Universal Robots PolyScope program: wrs2020_taskboard_belt.urp

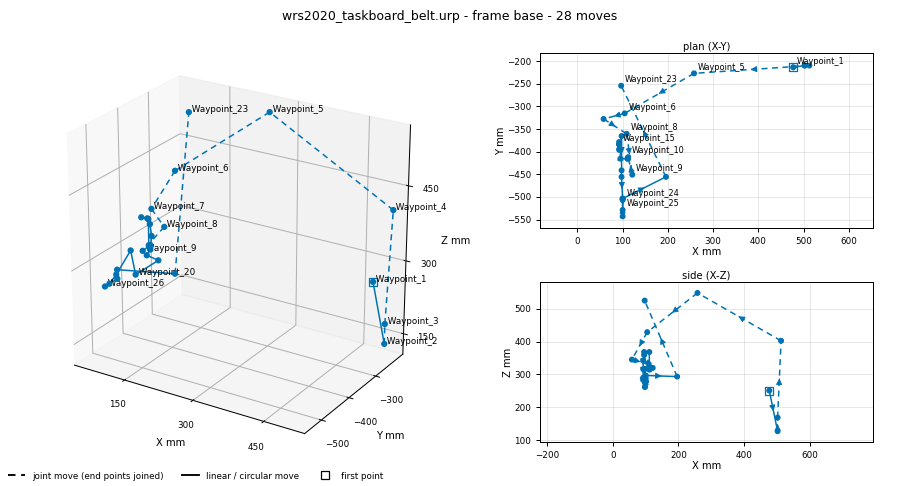
[picture p0: tool path of wrs2020_taskboard_belt.urp in frame base, 28 of 28 moves have a stored position in this frame; points joined in program order, loops and branches not executed]
Program wrs2020_taskboard_belt (installation=default directory=/programs/usbdisk createdIn=3.8.0.61336 lastSavedIn=3.8.0.61336 robotSerialNumber=2018357778)
Calibrated DH parameters: a=[0.000041, -0.391787, -0.374281, -0.000186, 0.000127, 0]; d=[0.08944, 27.652986, -9.436013, -18.1067, 0.094919, 0.082633]; alpha=[1.569511, -0.005996, -0.006449, 1.570544, -1.570475, 0]; deltaTheta=[0.000024, -0.400349, 0.096271, 0.298279, -0.00003, 0.000025]
Robot Program (runOnlyOnce=true)
  URCap Gripper (Robotiq_Grippers, Robotiq Inc.) dataModel(position=0.0, force=100.0, speed=100.0, positionInDouble=0.0, forceInDouble=100.0, speedInDouble=100.0, slaveIds=[9], blocking=true)
  MoveJ speed 60 deg/s, acceleration 80 deg/s^2 (useActiveTCP=true)
    Waypoint Waypoint_1: TCP in base x=476.88 y=-213.476 z=250.862 mm, rx=1.6793 ry=-1.6521 rz=-0.7958 rad; joints [147.47, -71.594, 89.892, -60.74, -116.873, 338.983] deg
  MoveL speed 250 mm/s, acceleration 1200 mm/s^2 (useActiveTCP=true) feature=Base
    Waypoint Waypoint_2: TCP in base x=502.313 y=-209.586 z=126.998 mm, rx=1.6772 ry=-1.66 rz=-0.8065 rad; joints [149.034, -61.436, 94.891, -75.152, -115.221, 340.261] deg
    URCap Gripper (Robotiq_Grippers, Robotiq Inc.) dataModel(position=100.0, force=100.0, speed=100.0, positionInDouble=100.0, forceInDouble=100.0, speedInDouble=100.0, slaveIds=[9], blocking=true)
  MoveJ speed 60 deg/s, acceleration 80 deg/s^2 (useActiveTCP=true)
    Waypoint Waypoint_3: TCP in base x=502.291 y=-209.619 z=168.566 mm, rx=1.6772 ry=-1.6602 rz=-0.8062 rad; joints [149.028, -64.302, 92.335, -69.737, -115.191, 340.279] deg
    Waypoint Waypoint_4: TCP in base x=512.821 y=-209.633 z=402.821 mm, rx=2.1959 ry=-2.1936 rz=-0.0165 rad; joints [146.25, -82.062, 85.641, -92.195, -92.332, 326.65] deg
    Waypoint Waypoint_5: TCP in base x=257.912 y=-226.881 z=548.602 mm, rx=-2.252 ry=-2.1409 rz=0.0571 rad; joints [120.027, -108.226, 87.388, -67.4, -92.623, 123.461] deg
    Popup Message (haltProgram=false message=waiting for a_bot to hold belt inputType=Text)
  MoveJ speed 60 deg/s, acceleration 80 deg/s^2 (useActiveTCP=true)
    Waypoint Waypoint_6: TCP in base x=104.652 y=-315.264 z=429.034 mm, rx=-0.7232 ry=-2.7798 rz=0.8385 rad; joints [93.055, -116.851, 119.471, -121.466, -107.654, 27.881] deg
    Waypoint Waypoint_7: TCP in base x=58.057 y=-327.656 z=345.432 mm, rx=-0.943 ry=-2.6822 rz=1.0186 rad; joints [84.311, -114.161, 133.07, -146.038, -105.388, 27.982] deg
  Popup Message (haltProgram=false message=wait for a_bot to move closer to pulley inputType=Text)
  MoveJ speed 60 deg/s, acceleration 80 deg/s^2 (useActiveTCP=true)
    Waypoint Waypoint_8: TCP in base x=109.129 y=-360.526 z=332.009 mm, rx=-1.6529 ry=-2.3933 rz=0.9597 rad; joints [95.219, -105.447, 127.131, -138.287, -116.294, 68.286] deg
    Waypoint Waypoint_9: TCP in base x=121.477 y=-450.838 z=319.976 mm, rx=-1.9847 ry=-2.0091 rz=0.7379 rad; joints [96.381, -91.245, 112.208, -119.67, -121.006, 93.458] deg
    Waypoint Waypoint_10: TCP in base x=112.095 y=-412.15 z=315.009 mm, rx=-1.9566 ry=-2.0028 rz=0.6969 rad; joints [95.734, -96.48, 117.235, -117.427, -121.063, 92.728] deg
  Popup Message (haltProgram=false message=wait for a_bot to finish placement inputType=Text)
  MoveL speed 250 mm/s, acceleration 1200 mm/s^2 (useActiveTCP=true) feature=Base
    Waypoint Waypoint_11: TCP in base x=111.067 y=-415.408 z=315.577 mm, rx=-1.9655 ry=-2.0043 rz=0.7162 rad; joints [95.563, -96.141, 117.17, -118.803, -121.129, 92.461] deg
    Waypoint Waypoint_12: TCP in base x=111.014 y=-415.438 z=368.385 mm, rx=-1.9655 ry=-2.004 rz=0.716 rad; joints [95.529, -98.391, 111.022, -110.38, -121.122, 92.491] deg
    Waypoint Waypoint_13: TCP in base x=95.213 y=-415.423 z=368.401 mm, rx=-1.9654 ry=-2.0041 rz=0.7161 rad; joints [93.34, -99.062, 111.894, -111.876, -120.787, 89.955] deg
    Waypoint Waypoint_14: TCP in base x=95.201 y=-395.921 z=359.198 mm, rx=-1.9656 ry=-2.0041 rz=0.7161 rad; joints [93.52, -101.499, 115.201, -112.651, -120.798, 90.156] deg
    Waypoint Waypoint_15: TCP in base x=92.395 y=-383.717 z=342.34 mm, rx=-1.9656 ry=-2.0041 rz=0.7163 rad; joints [93.226, -102.722, 118.728, -115.146, -120.743, 89.794] deg
    Waypoint Waypoint_16: TCP in base x=92.424 y=-378.74 z=316.285 mm, rx=-1.9655 ry=-2.0042 rz=0.7161 rad; joints [93.292, -102.186, 122.322, -119.247, -120.747, 89.837] deg
    Waypoint Waypoint_17: TCP in base x=92.37 y=-383.706 z=290.126 mm, rx=-1.9656 ry=-2.0041 rz=0.716 rad; joints [93.254, -99.843, 124.649, -123.945, -120.746, 89.776] deg
    Waypoint Waypoint_18: TCP in base x=92.376 y=-395.73 z=283.079 mm, rx=-1.9656 ry=-2.0041 rz=0.7161 rad; joints [93.151, -97.601, 123.978, -125.581, -120.74, 89.651] deg
    Waypoint Waypoint_19: TCP in base x=97.787 y=-365.382 z=262.233 mm, rx=-2.0667 ry=-2.0015 rz=0.9366 rad; joints [94.505, -99.478, 132.408, -142.318, -121.782, 90.846] deg
    Waypoint Waypoint_20: TCP in base x=97.788 y=-441.256 z=262.195 mm, rx=-2.0667 ry=-2.0016 rz=0.9364 rad; joints [93.65, -88.834, 122.921, -143.961, -121.543, 89.903] deg
    Waypoint Waypoint_21: TCP in base x=97.738 y=-455.581 z=316.933 mm, rx=-2.0668 ry=-2.0015 rz=0.9366 rad; joints [93.494, -91.095, 116.007, -134.854, -121.51, 89.794] deg
  MoveL speed 250 mm/s, acceleration 1200 mm/s^2 (useActiveTCP=true) feature=Base
    Waypoint Waypoint_24: TCP in base x=100.161 y=-506.631 z=288.366 mm, rx=-2.0669 ry=-2.0015 rz=0.9367 rad; joints [93.397, -82.486, 111.528, -139.056, -121.514, 89.661] deg
    Waypoint Waypoint_25: TCP in base x=100.189 y=-528.806 z=278.635 mm, rx=-2.0669 ry=-2.0015 rz=0.9367 rad; joints [93.244, -79.049, 109.068, -140.126, -121.477, 89.482] deg
    Waypoint Waypoint_26: TCP in base x=100.139 y=-542.854 z=278.562 mm, rx=-2.0669 ry=-2.0014 rz=0.9366 rad; joints [93.146, -77.333, 106.94, -139.76, -121.459, 89.381] deg
    Waypoint Waypoint_27: TCP in base x=100.153 y=-503.541 z=278.632 mm, rx=-2.0669 ry=-2.0013 rz=0.9368 rad; joints [93.423, -82.168, 112.794, -140.632, -121.525, 89.684] deg
    Waypoint Waypoint_28: TCP in base x=100.159 y=-503.538 z=296.982 mm, rx=-2.0669 ry=-2.0014 rz=0.9367 rad; joints [93.417, -83.468, 111.222, -137.751, -121.523, 89.695] deg
  MoveL speed 250 mm/s, acceleration 1200 mm/s^2 (useActiveTCP=true) feature=Base
    Waypoint Waypoint_22: TCP in base x=195.886 y=-455.587 z=293.483 mm, rx=-2.0667 ry=-2.0015 rz=0.9365 rad; joints [105.644, -85.473, 112.037, -128.892, -125.01, 103.726] deg
  MoveJ speed 60 deg/s, acceleration 80 deg/s^2 (useActiveTCP=true)
    Waypoint Waypoint_23: TCP in base x=96.884 y=-254.304 z=525.339 mm, rx=3.1071 ry=0.1116 rz=0.0373 rad; joints [85.767, -120.123, 98.055, -69.279, -88.529, 172.131] deg
